(* PLC project CoDeSys External Library Template, WAGO e!COCKPIT e!COCKPIT, author 3S - Smart Software Solutions GmbH *)
(* stored: creationDateTime 2019-10-29T12:37:19.313047, version 3.5.5.30, modificationDateTime 2019-10-29T12:36:39.3744516, organization 3S - Smart Software Solutions GmbH *)
(* Library project template with all possible element types, docu and a sample project structure *)

(* values of enumPPPSAnalizatorDirisA40Error: BrakKomunikacji: brak komunikacji z analizatorem; BrakZmianyParametrow: alarm braku zmiany wartości paramterów (napięcie, prąd) *)

(* Autor: Paweł Kąkol, 2018-09-04-PK Prawa majątkowe: Solwena Sp. z o.o., Aktualizacje: 2019-02-18-AWy: alarm braku zmiany wartości napięcia lub prądu Opis: fb służy do obsługi alarmów w fb analizatora sieci ECA0 na budynkach PPP Sopot (ENGIE) Diris A40 *)
{attribute 'qualified_only'}
{attribute 'strict'}
TYPE enumPPPSAnalizatorDirisA40Error : (BrakKomunikacji := 1, BrakZmianyParametrow := 2);
END_TYPE
